// TIA Portal V15.1 export
// export: Created 2024-05-17T05:38:59.6618517Z, ExportSetting WithDefaults, DisplayName Totally Integrated Automation Portal, DisplayVersion V15.1 Update 5, DisplayName TIA Portal Openness, DisplayVersion V15.1 Update 5, DisplayName SINAMICS Startdrive Advanced, DisplayVersion V15.1, DisplayName G130, G150, S120, S150, SINAMICS MV, S210, DisplayVersion V15.1, DisplayName G110M, G120, G120C, G120D, G120P, DisplayVersion V15.1, DisplayName STEP 7 Professional, DisplayVersion V15.1 Update 5, DisplayName STEP 7 Safety, DisplayVersion V15.1, DisplayName WinCC Professional, DisplayVersion V15.1 Update 5, DisplayName SIMATIC Visualization Architect, DisplayVersion V15.1
FUNCTION "209000NCP01Safety" : Void   // FC280, FBD
TITLE = 209000NCP01Safety
{ S7_Optimized_Access := 'FALSE' }
AUTHOR : VCC
VERSION : 0.1
// stored: AutoNumber false, IsIECCheckEnabled false, SetENOAutomatically False, UDAEnableTagReadback false
   VAR_OUTPUT
      O_AlarmA : Bool;   // Alarm A
      O_AlarmB : Bool;   // Alarm B
      O_AlarmC : Bool;   // Alarm C
      O_AlarmD : Bool;   // Alarm D
      O_AlarmABCondition : Bool;   // Alarms resetable
      H_IAnim : Word;   // Icon Animation
   END_VAR
BEGIN

REGION Network 1: **** 4.6 - Machine status - Indications **** Icon Animation
   // Icon animation
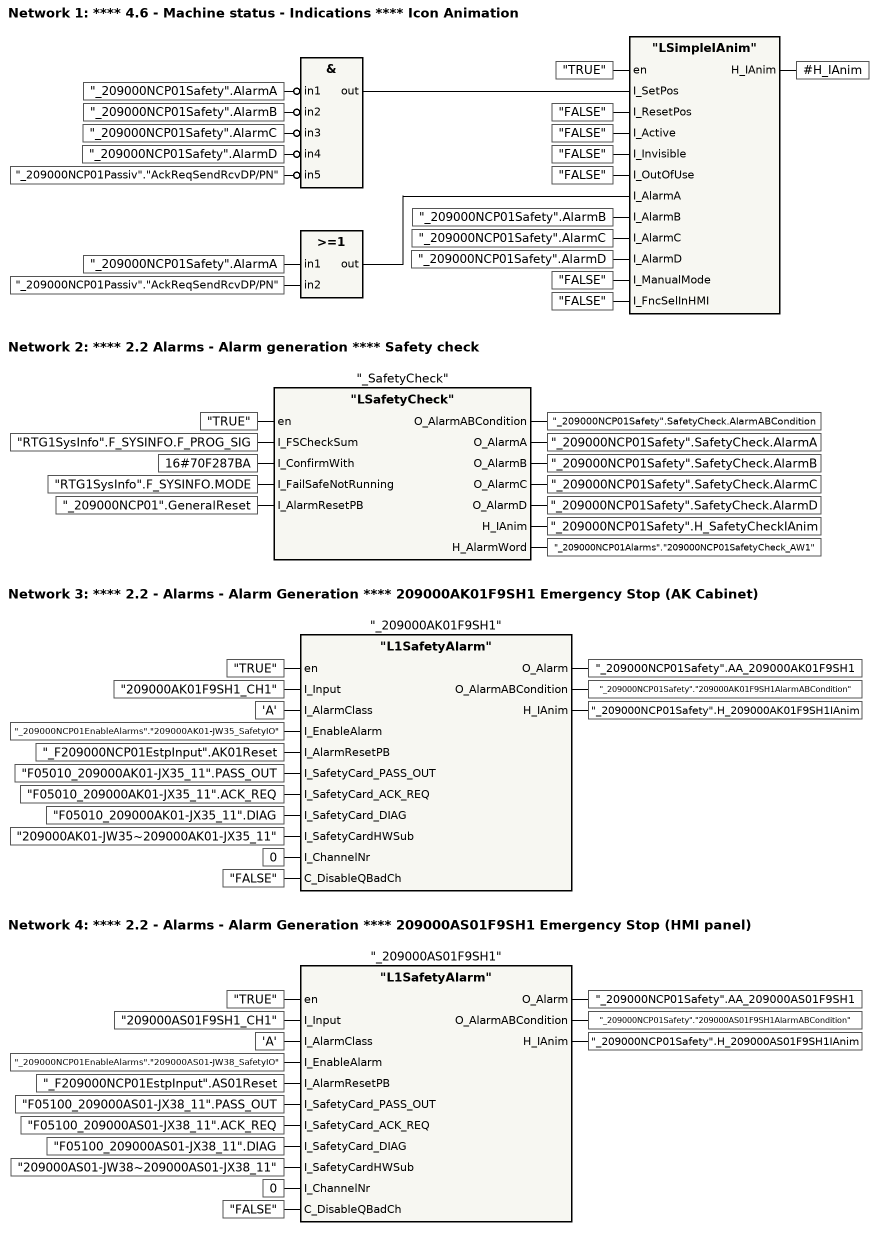
   IF "TRUE" THEN
       "LSimpleIAnim"(I_SetPos := NOT "_209000NCP01Safety".AlarmA AND NOT "_209000NCP01Safety".AlarmB AND NOT "_209000NCP01Safety".AlarmC AND NOT "_209000NCP01Safety".AlarmD AND NOT "_209000NCP01Passiv"."AckReqSendRcvDP/PN",
                      I_ResetPos := "FALSE",
                      I_Active := "FALSE",
                      I_Invisible := "FALSE",
                      I_OutOfUse := "FALSE",
                      I_AlarmA := "_209000NCP01Safety".AlarmA OR "_209000NCP01Passiv"."AckReqSendRcvDP/PN",
                      I_AlarmB := "_209000NCP01Safety".AlarmB,
                      I_AlarmC := "_209000NCP01Safety".AlarmC,
                      I_AlarmD := "_209000NCP01Safety".AlarmD,
                      I_ManualMode := "FALSE",
                      I_FncSelInHMI := "FALSE",
                      H_IAnim => #H_IAnim);
   END_IF;
END_REGION

REGION Network 2: **** 2.2 Alarms - Alarm generation **** Safety check
   // Safety check
   IF "TRUE" THEN
       "_SafetyCheck"(I_FSCheckSum := "RTG1SysInfo".F_SYSINFO.F_PROG_SIG,   // "LSafetyCheck"
                      I_ConfirmWith := 16#70F287BA,
                      I_FailSafeNotRunning := "RTG1SysInfo".F_SYSINFO.MODE,
                      I_AlarmResetPB := "_209000NCP01".GeneralReset,
                      O_AlarmABCondition => "_209000NCP01Safety".SafetyCheck.AlarmABCondition,
                      O_AlarmA => "_209000NCP01Safety".SafetyCheck.AlarmA,
                      O_AlarmB => "_209000NCP01Safety".SafetyCheck.AlarmB,
                      O_AlarmC => "_209000NCP01Safety".SafetyCheck.AlarmC,
                      O_AlarmD => "_209000NCP01Safety".SafetyCheck.AlarmD,
                      H_IAnim => "_209000NCP01Safety".H_SafetyCheckIAnim,
                      H_AlarmWord => "_209000NCP01Alarms"."209000NCP01SafetyCheck_AW1");
   END_IF;
END_REGION

REGION Network 3: **** 2.2 - Alarms - Alarm Generation **** 209000AK01F9SH1 Emergency Stop (AK Cabinet)
   // Emergency Stop
   IF "TRUE" THEN
       "_209000AK01F9SH1"(I_Input := "209000AK01F9SH1_CH1",   // "L1SafetyAlarm"
                          I_AlarmClass := 'A',
                          I_EnableAlarm := "_209000NCP01EnableAlarms"."209000AK01-JW35_SafetyIO",
                          I_AlarmResetPB := "_F209000NCP01EstpInput".AK01Reset,
                          I_SafetyCard_PASS_OUT := "F05010_209000AK01-JX35_11".PASS_OUT,
                          I_SafetyCard_ACK_REQ := "F05010_209000AK01-JX35_11".ACK_REQ,
                          I_SafetyCard_DIAG := "F05010_209000AK01-JX35_11".DIAG,
                          I_SafetyCardHWSub := "209000AK01-JW35~209000AK01-JX35_11",
                          I_ChannelNr := 0,
                          C_DisableQBadCh := "FALSE",
                          O_Alarm => "_209000NCP01Safety".AA_209000AK01F9SH1,
                          O_AlarmABCondition => "_209000NCP01Safety"."209000AK01F9SH1AlarmABCondition",
                          H_IAnim => "_209000NCP01Safety".H_209000AK01F9SH1IAnim);
   END_IF;
END_REGION

REGION Network 4: **** 2.2 - Alarms - Alarm Generation **** 209000AS01F9SH1 Emergency Stop (HMI panel)
   // Emergency Stop
   IF "TRUE" THEN
       "_209000AS01F9SH1"(I_Input := "209000AS01F9SH1_CH1",   // "L1SafetyAlarm"
                          I_AlarmClass := 'A',
                          I_EnableAlarm := "_209000NCP01EnableAlarms"."209000AS01-JW38_SafetyIO",
                          I_AlarmResetPB := "_F209000NCP01EstpInput".AS01Reset,
                          I_SafetyCard_PASS_OUT := "F05100_209000AS01-JX38_11".PASS_OUT,
                          I_SafetyCard_ACK_REQ := "F05100_209000AS01-JX38_11".ACK_REQ,
                          I_SafetyCard_DIAG := "F05100_209000AS01-JX38_11".DIAG,
                          I_SafetyCardHWSub := "209000AS01-JW38~209000AS01-JX38_11",
                          I_ChannelNr := 0,
                          C_DisableQBadCh := "FALSE",
                          O_Alarm => "_209000NCP01Safety".AA_209000AS01F9SH1,
                          O_AlarmABCondition => "_209000NCP01Safety"."209000AS01F9SH1AlarmABCondition",
                          H_IAnim => "_209000NCP01Safety".H_209000AS01F9SH1IAnim);
   END_IF;
END_REGION

REGION Network 5: **** 2.2 - Alarms - Alarm Generation **** 209000AS02F9SH1 Emergency Stop (HMI panel)
   // Emergency Stop
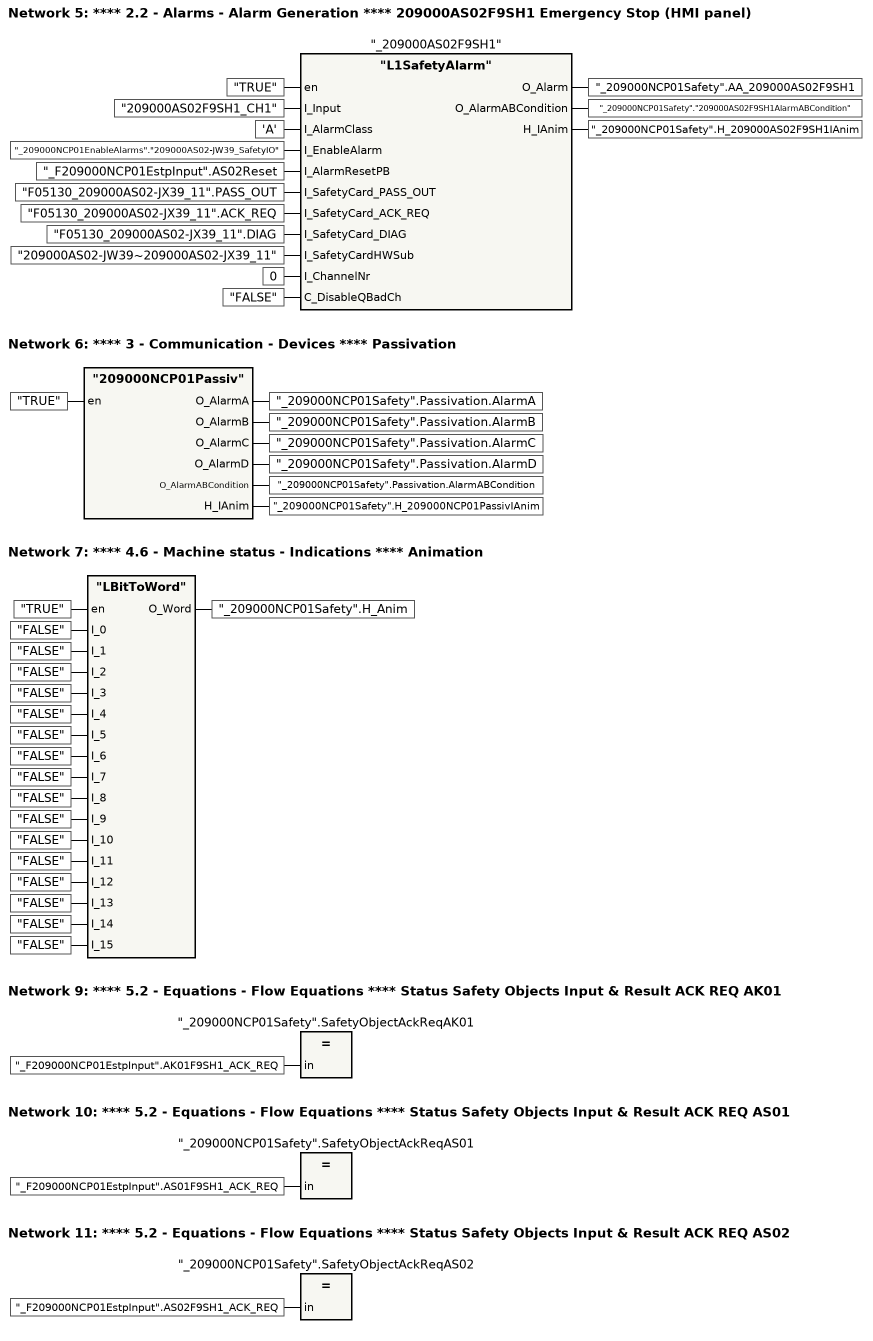
   IF "TRUE" THEN
       "_209000AS02F9SH1"(I_Input := "209000AS02F9SH1_CH1",   // "L1SafetyAlarm"
                          I_AlarmClass := 'A',
                          I_EnableAlarm := "_209000NCP01EnableAlarms"."209000AS02-JW39_SafetyIO",
                          I_AlarmResetPB := "_F209000NCP01EstpInput".AS02Reset,
                          I_SafetyCard_PASS_OUT := "F05130_209000AS02-JX39_11".PASS_OUT,
                          I_SafetyCard_ACK_REQ := "F05130_209000AS02-JX39_11".ACK_REQ,
                          I_SafetyCard_DIAG := "F05130_209000AS02-JX39_11".DIAG,
                          I_SafetyCardHWSub := "209000AS02-JW39~209000AS02-JX39_11",
                          I_ChannelNr := 0,
                          C_DisableQBadCh := "FALSE",
                          O_Alarm => "_209000NCP01Safety".AA_209000AS02F9SH1,
                          O_AlarmABCondition => "_209000NCP01Safety"."209000AS02F9SH1AlarmABCondition",
                          H_IAnim => "_209000NCP01Safety".H_209000AS02F9SH1IAnim);
   END_IF;
END_REGION

REGION Network 6: **** 3 - Communication - Devices **** Passivation
   // Passivation
   IF "TRUE" THEN
       "209000NCP01Passiv"(O_AlarmA => "_209000NCP01Safety".Passivation.AlarmA,
                           O_AlarmB => "_209000NCP01Safety".Passivation.AlarmB,
                           O_AlarmC => "_209000NCP01Safety".Passivation.AlarmC,
                           O_AlarmD => "_209000NCP01Safety".Passivation.AlarmD,
                           O_AlarmABCondition => "_209000NCP01Safety".Passivation.AlarmABCondition,
                           H_IAnim => "_209000NCP01Safety".H_209000NCP01PassivIAnim);
   END_IF;
END_REGION

REGION Network 7: **** 4.6 - Machine status - Indications **** Animation
   // Animation
   IF "TRUE" THEN
       "LBitToWord"(I_0 := "FALSE",
                    I_1 := "FALSE",
                    I_2 := "FALSE",
                    I_3 := "FALSE",
                    I_4 := "FALSE",
                    I_5 := "FALSE",
                    I_6 := "FALSE",
                    I_7 := "FALSE",
                    I_8 := "FALSE",
                    I_9 := "FALSE",
                    I_10 := "FALSE",
                    I_11 := "FALSE",
                    I_12 := "FALSE",
                    I_13 := "FALSE",
                    I_14 := "FALSE",
                    I_15 := "FALSE",
                    O_Word => "_209000NCP01Safety".H_Anim);
   END_IF;
END_REGION

NETWORK
TITLE = **** 4.6 - Machine Status - Indications **** Animation DB number
// DB number
      OPN   "_209000NCP01Safety";
      L     DBNO;
      T     "_209000NCP01Safety".H_DBnr;

REGION Network 9: **** 5.2 - Equations - Flow Equations **** Status Safety Objects Input & Result ACK REQ AK01
   // AK
   "_209000NCP01Safety".SafetyObjectAckReqAK01 := "_F209000NCP01EstpInput".AK01F9SH1_ACK_REQ;
END_REGION

REGION Network 10: **** 5.2 - Equations - Flow Equations **** Status Safety Objects Input & Result ACK REQ AS01
   // AS
   "_209000NCP01Safety".SafetyObjectAckReqAS01 := "_F209000NCP01EstpInput".AS01F9SH1_ACK_REQ;
END_REGION

REGION Network 11: **** 5.2 - Equations - Flow Equations **** Status Safety Objects Input & Result ACK REQ AS02
   // AS
   "_209000NCP01Safety".SafetyObjectAckReqAS02 := "_F209000NCP01EstpInput".AS02F9SH1_ACK_REQ;
END_REGION

REGION Network 12: **** 9 - Alarm Summary **** Alarm AB condition
   // Alarm AB condition
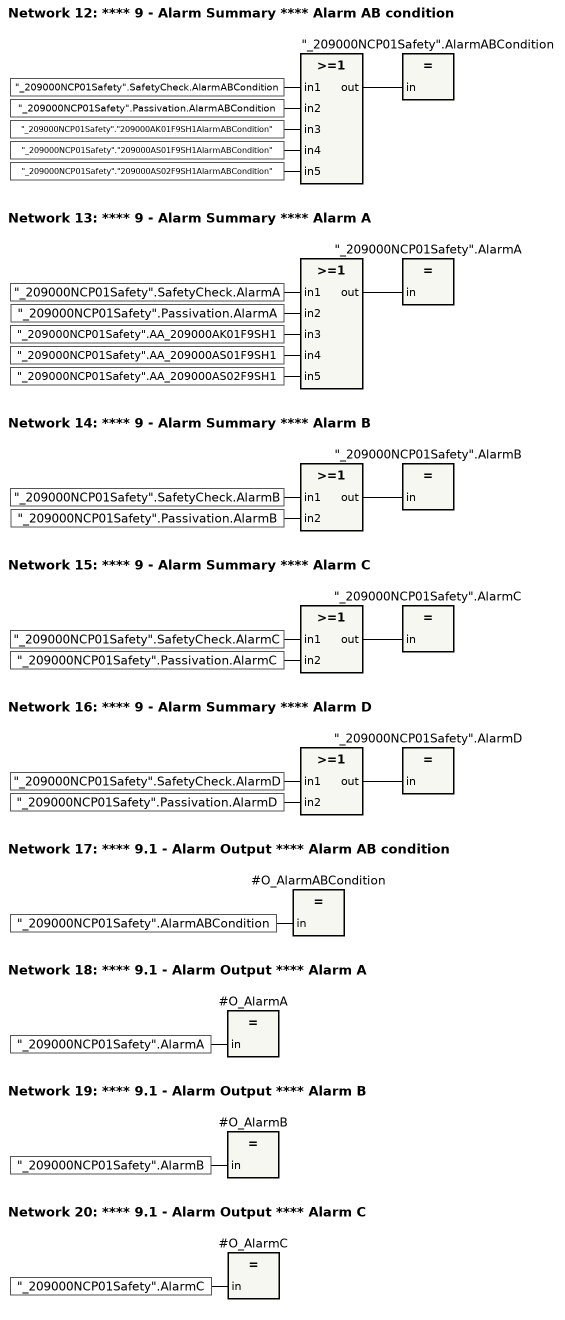
   "_209000NCP01Safety".AlarmABCondition := "_209000NCP01Safety".SafetyCheck.AlarmABCondition OR "_209000NCP01Safety".Passivation.AlarmABCondition OR "_209000NCP01Safety"."209000AK01F9SH1AlarmABCondition" OR "_209000NCP01Safety"."209000AS01F9SH1AlarmABCondition" OR "_209000NCP01Safety"."209000AS02F9SH1AlarmABCondition";
END_REGION

REGION Network 13: **** 9 - Alarm Summary **** Alarm A
   // Summary of alarms A
   "_209000NCP01Safety".AlarmA := "_209000NCP01Safety".SafetyCheck.AlarmA OR "_209000NCP01Safety".Passivation.AlarmA OR "_209000NCP01Safety".AA_209000AK01F9SH1 OR "_209000NCP01Safety".AA_209000AS01F9SH1 OR "_209000NCP01Safety".AA_209000AS02F9SH1;
END_REGION

REGION Network 14: **** 9 - Alarm Summary **** Alarm B
   // Summary of alarms B
   "_209000NCP01Safety".AlarmB := "_209000NCP01Safety".SafetyCheck.AlarmB OR "_209000NCP01Safety".Passivation.AlarmB;
END_REGION

REGION Network 15: **** 9 - Alarm Summary **** Alarm C
   // Summary of alarms C
   "_209000NCP01Safety".AlarmC := "_209000NCP01Safety".SafetyCheck.AlarmC OR "_209000NCP01Safety".Passivation.AlarmC;
END_REGION

REGION Network 16: **** 9 - Alarm Summary **** Alarm D
   // Summary of alarms D
   "_209000NCP01Safety".AlarmD := "_209000NCP01Safety".SafetyCheck.AlarmD OR "_209000NCP01Safety".Passivation.AlarmD;
END_REGION

REGION Network 17: **** 9.1 - Alarm Output **** Alarm AB condition
   // Alarm AB condition
   #O_AlarmABCondition := "_209000NCP01Safety".AlarmABCondition;
END_REGION

REGION Network 18: **** 9.1 - Alarm Output **** Alarm A
   // Summary of alarms A
   #O_AlarmA := "_209000NCP01Safety".AlarmA;
END_REGION

REGION Network 19: **** 9.1 - Alarm Output **** Alarm B
   // Summary of alarms B
   #O_AlarmB := "_209000NCP01Safety".AlarmB;
END_REGION

REGION Network 20: **** 9.1 - Alarm Output **** Alarm C
   // Summary of alarms C
   #O_AlarmC := "_209000NCP01Safety".AlarmC;
END_REGION

REGION Network 21: **** 9.1 - Alarm Output **** Alarm D
   // Summary of alarms D
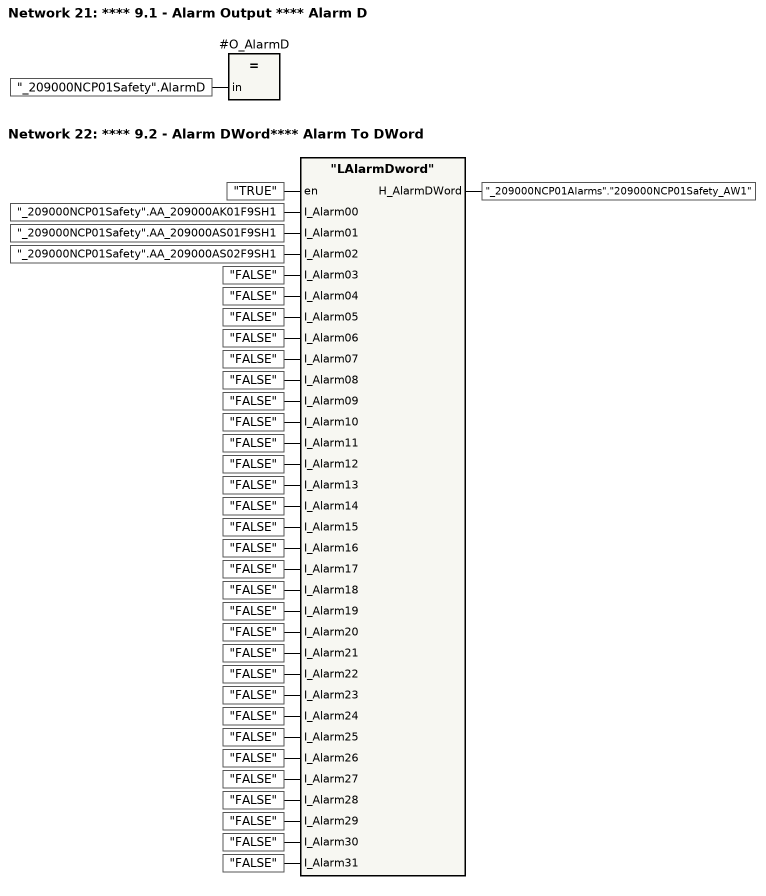
   #O_AlarmD := "_209000NCP01Safety".AlarmD;
END_REGION

REGION Network 22: **** 9.2 - Alarm DWord**** Alarm To DWord
   // Alarm Word
   IF "TRUE" THEN
       "LAlarmDword"(I_Alarm00 := "_209000NCP01Safety".AA_209000AK01F9SH1,
                     I_Alarm01 := "_209000NCP01Safety".AA_209000AS01F9SH1,
                     I_Alarm02 := "_209000NCP01Safety".AA_209000AS02F9SH1,
                     I_Alarm03 := "FALSE",
                     I_Alarm04 := "FALSE",
                     I_Alarm05 := "FALSE",
                     I_Alarm06 := "FALSE",
                     I_Alarm07 := "FALSE",
                     I_Alarm08 := "FALSE",
                     I_Alarm09 := "FALSE",
                     I_Alarm10 := "FALSE",
                     I_Alarm11 := "FALSE",
                     I_Alarm12 := "FALSE",
                     I_Alarm13 := "FALSE",
                     I_Alarm14 := "FALSE",
                     I_Alarm15 := "FALSE",
                     I_Alarm16 := "FALSE",
                     I_Alarm17 := "FALSE",
                     I_Alarm18 := "FALSE",
                     I_Alarm19 := "FALSE",
                     I_Alarm20 := "FALSE",
                     I_Alarm21 := "FALSE",
                     I_Alarm22 := "FALSE",
                     I_Alarm23 := "FALSE",
                     I_Alarm24 := "FALSE",
                     I_Alarm25 := "FALSE",
                     I_Alarm26 := "FALSE",
                     I_Alarm27 := "FALSE",
                     I_Alarm28 := "FALSE",
                     I_Alarm29 := "FALSE",
                     I_Alarm30 := "FALSE",
                     I_Alarm31 := "FALSE",
                     H_AlarmDWord => "_209000NCP01Alarms"."209000NCP01Safety_AW1");
   END_IF;
END_REGION
END_FUNCTION
